TYPE APP_Com :
STRUCT
	bBackStationPosFinish:BOOL;
	bBendStationPosFinish:BOOL;
END_STRUCT
END_TYPE

(* stored: Version 1.1.0.1, ProductVersion 3.1.4024.12
   DUT APP_Com: Id {2110ab18-2401-4132-917e-be77e5ebb47b} *)
